FUNCTION_BLOCK EthercatMasterAdditionalSyncUnit EXTENDS EthercatMasterBase
VAR
	AdditionalSyncUnit : SyncUnit;
	AdditionalSyncUnitHadIssue : BOOL;
END_VAR

METHOD Diagnostics
VAR
    _deviceStatus : EthercatMasterDeviceStatus;
    _i : UINT;
    _tmpString : STRING(125);
    _tmpErrorMessage : STRING(125);
END_VAR
IF AdditionalSyncUnit.HasIssue THEN
	SUPER^.AdditionalSyncUnitHasIssue := TRUE;
END_IF

IF AdditionalSyncUnitHadIssue AND NOT AdditionalSyncUnit.HasIssue THEN
	SUPER^.AdditionalSyncUnitHasIssue := FALSE;
END_IF

AdditionalSyncUnitHadIssue := AdditionalSyncUnit.HasIssue;

SUPER^.Diagnostics();
END_METHOD

END_FUNCTION_BLOCK

(* stored: Version 1.1.0.1, ProductVersion 3.1.4024.9
   POU EthercatMasterAdditionalSyncUnit: Id {527bad92-3897-0c10-1da2-1e462ac8b901}, SpecialFunc None
   Method Diagnostics: Id {f4e97dcc-80b0-0ba3-2d1f-3e774944ff62} *)
